{attribute 'GeneratedUsingTerminal: EPP2038-0001-0016'}
{attribute addProperty BoxType "EPP2038-0001-0016"}
{attribute addProperty Id "Diag_Channel_1AT %I*Diag_Channel_830843C11Diag_Channel_2AT %I*Diag_Channel_830843C11Diag_Channel_3AT %I*Diag_Channel_830843C11Diag_Channel_4AT %I*Diag_Channel_830843C11Diag_Channel_5AT %I*Diag_Channel_830843C11Diag_Channel_6AT %I*Diag_Channel_830843C11Diag_Channel_7AT %I*Diag_Channel_830843C11Diag_Channel_8AT %I*Diag_Channel_830843C11Channel_1AT %Q*Channel_42CA91F71Channel_2AT %Q*Channel_42CA91F71Channel_3AT %Q*Channel_42CA91F71Channel_4AT %Q*Channel_42CA91F71Channel_5AT %Q*Channel_42CA91F71Channel_6AT %Q*Channel_42CA91F71Channel_7AT %Q*Channel_42CA91F71Channel_8AT %Q*Channel_42CA91F71WcStateAT %I*WcState_9091E0EB2InfoDataAT %I*InfoData_6F19DB2B2"}
{attribute addProperty CRC "987827671"}
{attribute addProperty Size "20"}
TYPE EPP2038_3AE10DD7 EXTENDS EtcSlaveTerminalBase_947E5A46 :
STRUCT
	{attribute addProperty Name "Diag_Channel_1"}
	Diag_Channel_1 : Diag_Channel_830843C1;
	{attribute addProperty Name "Diag_Channel_2"}
	Diag_Channel_2 : Diag_Channel_830843C1;
	{attribute addProperty Name "Diag_Channel_3"}
	Diag_Channel_3 : Diag_Channel_830843C1;
	{attribute addProperty Name "Diag_Channel_4"}
	Diag_Channel_4 : Diag_Channel_830843C1;
	{attribute addProperty Name "Diag_Channel_5"}
	Diag_Channel_5 : Diag_Channel_830843C1;
	{attribute addProperty Name "Diag_Channel_6"}
	Diag_Channel_6 : Diag_Channel_830843C1;
	{attribute addProperty Name "Diag_Channel_7"}
	Diag_Channel_7 : Diag_Channel_830843C1;
	{attribute addProperty Name "Diag_Channel_8"}
	Diag_Channel_8 : Diag_Channel_830843C1;
	{attribute addProperty Name "Channel_1"}
	Channel_1 : Channel_42CA91F7;
	{attribute addProperty Name "Channel_2"}
	Channel_2 : Channel_42CA91F7;
	{attribute addProperty Name "Channel_3"}
	Channel_3 : Channel_42CA91F7;
	{attribute addProperty Name "Channel_4"}
	Channel_4 : Channel_42CA91F7;
	{attribute addProperty Name "Channel_5"}
	Channel_5 : Channel_42CA91F7;
	{attribute addProperty Name "Channel_6"}
	Channel_6 : Channel_42CA91F7;
	{attribute addProperty Name "Channel_7"}
	Channel_7 : Channel_42CA91F7;
	{attribute addProperty Name "Channel_8"}
	Channel_8 : Channel_42CA91F7;
	{attribute addProperty Name "WcState"}
	WcState : WcState_9091E0EB;
	{attribute addProperty Name "InfoData"}
	InfoData : InfoData_6F19DB2B;
END_STRUCT
END_TYPE

(* stored: Version 1.2.0.0, ProductVersion 3.1.4024.9
   DUT EPP2038_3AE10DD7: Id {5857660b-34b0-4b6f-94cf-319a7034b910} *)
